{attribute 'GeneratedUsingTerminal: EL3783-0000-0018'}
{attribute addProperty BoxType "EL3783-0000-0018"}
{attribute addProperty Id "I1_SamplesAT %I*I1_Samples_1109DCAA40"}
{attribute addProperty CRC "2003392412"}
{attribute addProperty Size "40"}
TYPE L1_Current_Samples_7769579C :
STRUCT
	{attribute addProperty Name "I1_Samples"}
	I1_Samples AT %I* : I1_Samples_1109DCAA;
END_STRUCT
END_TYPE

(* stored: Version 1.2.0.0, ProductVersion 3.1.4024.9
   DUT L1_Current_Samples_7769579C: Id {c58d56bb-aa89-4da7-a6f0-c76da2863ee5} *)
